FUNCTION putUint : BOOL
	VAR_INPUT
		uintVar : UINT;
	END_VAR
	VAR_IN_OUT
		bufferRef : POINTER TO USINT;
	END_VAR

memcpy(bufferRef, ADR(uintVar), SIZEOF(UINT));
bufferRef := bufferRef + SIZEOF(UINT);
putUint := TRUE;

END_FUNCTION

(* stored: Version 1.1.0.1, ProductVersion 3.1.4024.3
   POU putUint: Id {0797683a-1211-018e-1d9c-09e54da39ce9}, SpecialFunc None *)
